TYPE ST_PU_Schuetz_Zustand :
STRUCT
	Betrieb_Anford	: BOOL;
	Betrieb_Soll		: BOOL;
	Betrieb			: BOOL;

	Freigabe			: BOOL;
	Freigabe_Deakt	: BOOL;
	Freigabe_Code	: WORD;

	Stoerung			: BOOL;
	Stoerung_Code	: WORD;

	Warnung			: BOOL;
	Warnung_Code	: WORD;

	Quittierung		: BOOL;

	Status			: SINT;
	Status_Vorl		: BOOL;
	Status_Nachl		: BOOL;
END_STRUCT
END_TYPE

(* stored: Version 1.1.0.1, ProductVersion 3.1.4024.9
   DUT ST_PU_Schuetz_Zustand: Id {ccf5edb2-f62e-47dd-8b1d-11c43ea9c21e} *)
